FUNCTION_BLOCK Aborting IMPLEMENTS ITF_PackMLState
VAR
END_VAR

METHOD CyclicLogic : BOOL
VAR_INPUT
END_VAR
END_METHOD

{warning 'add method implementation '}
METHOD EStop : BOOL
END_METHOD

{warning 'add method implementation '}
METHOD Reset : BOOL
END_METHOD

{warning 'add method implementation '}
METHOD SetContext : BOOL
VAR_INPUT
	context	: REFERENCE TO SomeMachine;
END_VAR
END_METHOD

{warning 'add method implementation '}
METHOD Start : BOOL
END_METHOD

{warning 'add method implementation '}
METHOD Stop : BOOL
END_METHOD

END_FUNCTION_BLOCK

(* stored: Version 1.1.0.1, ProductVersion 3.1.4024.12
   POU Aborting: Id {53b868d1-8bc9-4c10-8ac2-c1d64eeae366}, SpecialFunc None
   Method CyclicLogic: Id {6c0f6590-0459-482e-8713-8ce383ea8165}
   Method EStop: Id {60859f9c-407e-4ad8-a2cc-ce6c27e8996f}
   Method Reset: Id {2650164a-692b-43b9-9794-739b4238b555}
   Method SetContext: Id {44eb273c-3e24-4070-b0da-a59f6767b731}
   Method Start: Id {006918a1-0058-4df6-83fd-6a4309e2c2e0}
   Method Stop: Id {4f8d02bb-0009-4525-8978-3b46006ea160} *)
